// TIA Portal V16 export
// export: Created 2021-08-10T09:05:00.1028573Z, ExportSetting WithDefaults, WithReadOnly, DisplayName Totally Integrated Automation Portal, DisplayVersion V16, DisplayName TIA Portal Version Control Interface, DisplayVersion V16, DisplayName TIA Portal Openness, DisplayVersion V16, DisplayName TIA Portal Teamcenter Gateway, DisplayVersion V16, DisplayName SINAMICS Startdrive Advanced, DisplayVersion V16, DisplayName SINAMICS Startdrive G130, G150, S120, S150, SINAMICS MV, S210, DisplayVersion V16, DisplayName SINAMICS Startdrive G110M, G120, G120C, G120D, G120P, DisplayVersion V16, DisplayName STEP 7 Professional, DisplayVersion V16, DisplayName STEP 7 Safety, DisplayVersion V16, DisplayName WinCC Unified SCADA Engineering System, DisplayVersion V16
FUNCTION "fcHMIBitEnable" : Void   // FC329, FBD
TITLE = Handles an async reading of an HMI bit to avoid race conditions, includes an enable bit
{ S7_Optimized_Access := 'TRUE' }
VERSION : 0.1
// stored: AutoNumber true, CodeModifiedDate 2020-08-01T14:00:25.8449031Z, CompileDate 2021-07-03T08:38:37.4904384Z, CreationDate 2020-02-26T07:34:28.9567791Z, HandleErrorsWithinBlock false, InterfaceModifiedDate 2017-10-26T17:33:11.2112674Z, IsConsistent true, IsIECCheckEnabled false, IsKnowHowProtected false, IsWriteProtected false, LibraryConformanceStatus The object is library-conformant., LibraryType fcHMIBitEnable V 3.0.3, LibraryTypeVersionGuid be26d641-fc92-415f-8b4f-76383b13c227, ModifiedDate 2020-08-01T14:00:32.9533133Z, ParameterModified 2017-10-26T17:33:11.2112674Z, PLCSimAdvancedSupport true, SetENOAutomatically false, StructureModified 2017-10-26T17:33:11.2112674Z, UDAEnableTagReadback false
   VAR_INPUT
      bInToggle : Bool;
      bInLatch : Bool;
      bInEnable : Bool;
   END_VAR
   VAR_OUTPUT
      bOutEnable : Bool;
   END_VAR
   VAR_IN_OUT
      bInOutHMI : Bool;
      bInOutPLC : Bool;
   END_VAR
   VAR_TEMP   // added for the SCL form of the ladder/FBD networks
      _w1 : Bool;
   END_VAR
BEGIN

REGION Network 1: If not latching or toggling, reset the PLC bit every scan
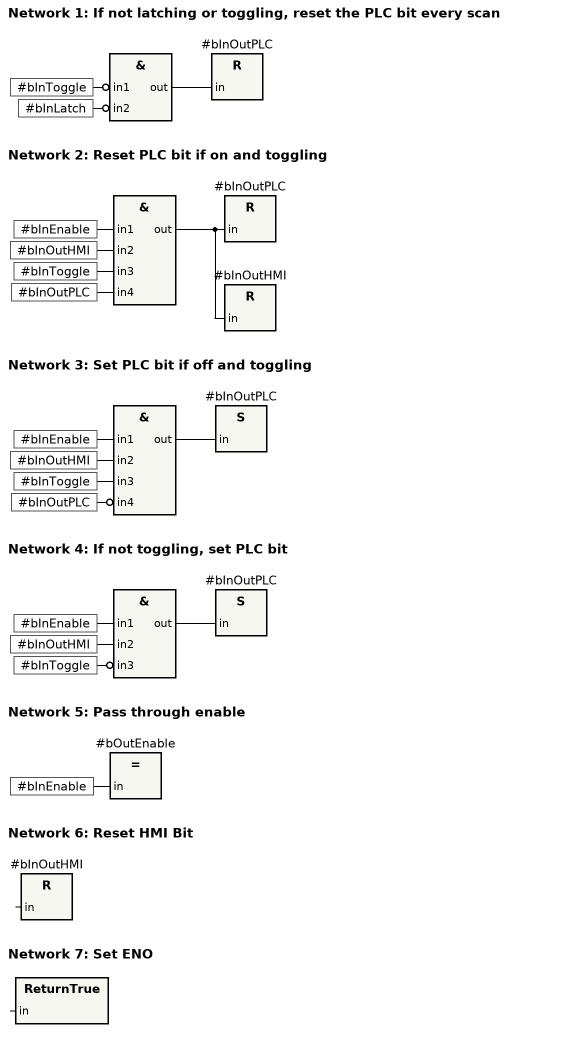
   IF NOT #bInToggle AND NOT #bInLatch THEN #bInOutPLC := FALSE; END_IF;
END_REGION

REGION Network 2: Reset PLC bit if on and toggling
   #_w1 := #bInEnable AND #bInOutHMI AND #bInToggle AND #bInOutPLC;
   IF #_w1 THEN
       #bInOutPLC := FALSE;
       #bInOutHMI := FALSE;
   END_IF;
END_REGION

REGION Network 3: Set PLC bit if off and toggling
   IF #bInEnable AND #bInOutHMI AND #bInToggle AND NOT #bInOutPLC THEN #bInOutPLC := TRUE; END_IF;
END_REGION

REGION Network 4: If not toggling, set PLC bit
   IF #bInEnable AND #bInOutHMI AND NOT #bInToggle THEN #bInOutPLC := TRUE; END_IF;
END_REGION

REGION Network 5: Pass through enable
   #bOutEnable := #bInEnable;
END_REGION

REGION Network 6: Reset HMI Bit
   #bInOutHMI := FALSE;
END_REGION

REGION Network 7: Set ENO
   ENO := TRUE;
   RETURN;
END_REGION
END_FUNCTION
